PROGRAM MAIN
VAR
	bOperationMode	: BOOL; // False:Manual, True:RecipeControl

	bTest1 : BOOL;
	bTest2 : BOOL;
	bTest3 : BOOL;
END_VAR

(* Modify Program *)

P11_E3508(); //Temp Controller
P12_IQ_PLUS(); //Throttle Valve Controller
P13_LineHeater();
P14_ThermalBath();
P15_RotationOperation();
P16_CoverOperation();
P17_DOROperation();
P20_BackgroundCom();
P21_Background_LineHeater();
P22_Background_ThermalBath();
P22_Background_ThermalBath();

IF NOT(bOperationMode) THEN
	P30_ManualControl(); //매뉴얼 콘트롤
ELSE
	P50_RecipeControl(); //레시피 콘트론
END_IF

P70_Interface();
P90_Interlock();
P91_Monitoring();
P92_Maintenance();

bTest1 := GVL_IO.aInputState[1].12;
bTest2 := GVL_IO.aInputState[1].13;
bTest3 := GVL_IO.aInputState[1].14;
(* Interlock Condtion *)
// DOR Operation Condition

END_PROGRAM

(* stored: Version 1.1.0.1, ProductVersion 3.1.4026.11
   POU MAIN: Id {c65bb020-a024-43e6-87d0-b2b9cfee7c16}, SpecialFunc None *)
